TYPE "udtAnalogInput"
VERSION : 0.1
   STRUCT
      rLowCalibration : Real;
      rHighCalibration : Real;
      rRawValue : Int;
      rActual : Real;
   END_STRUCT;

END_TYPE

